{attribute 'linkalways'} 
{attribute 'no_explicit_call' := 'This FB is a CLASS and must be accessed using methods or properties'}
{attribute 'enable_dynamic_creation'}
FUNCTION_BLOCK _TcVnRectangle EXTENDS AliasDatatypeBase
VAR
	localData : TcVnRectangle;
	activeData : REFERENCE TO TcVnRectangle REF= localData;
	aliasBaseDatatype : _TcVnRectangle_DINT;
END_VAR

PROPERTY PUBLIC Address : PVOID
GET
Address := ADR(activeData);
END_GET
END_PROPERTY

METHOD PUBLIC ClearReference
VAR_INPUT
END_VAR
activeData REF= localData;
SetBaseDatatypeReference();
END_METHOD

METHOD PUBLIC Clone : I_Datatype
VAR
    pClone : POINTER TO _TcVnRectangle;
END_VAR
pClone := __NEW(_TcVnRectangle);
Clone := pClone^;
END_METHOD

METHOD FB_init : BOOL
VAR_INPUT
	bInitRetains : BOOL; // if TRUE, the retain variables are initialized (warm start / cold start)
	bInCopyCode : BOOL;  // if TRUE, the instance afterwards gets moved into the copy code (online change)
	//InitialValue : <type>; // if possible, not all values can be initialized
END_VAR
//localData := InitialValue; // if possible, not all values can be initialized
SetBaseDatatypeReference();
AddBaseDatatype(aliasBaseDatatype);
END_METHOD

PROPERTY PUBLIC Identifier : T_MAXSTRING
GET
Identifier := 'TcVnRectangle';
END_GET
END_PROPERTY

METHOD PUBLIC MakeReferenceTo
VAR_INPUT
	ReferenceTarget : REFERENCE TO TcVnRectangle_DINT;
END_VAR
activeData REF= ReferenceTarget;
SetBaseDatatypeReference();
END_METHOD

METHOD PROTECTED SetBaseDatatypeReference
VAR_INPUT
END_VAR
aliasBaseDatatype.MakeReferenceTo(activeData);
END_METHOD

PROPERTY PUBLIC Size : UDINT
GET
Size := SIZEOF(activeData);
END_GET
END_PROPERTY

METHOD TryMakeReferenceTo : BOOL
VAR_INPUT
	Target : I_Datatype;
END_VAR
VAR
	targetAsAlias : I_AliasDatatype;
	pTargetData : POINTER TO TcVnRectangle_DINT;
END_VAR
IF NOT Target.TryResolveAsAliasDatatype(targetAsAlias) THEN
	RETURN;
END_IF

IF targetAsAlias.Identifier <> Identifier THEN
	RETURN;
END_IF

pTargetData := Target.Address;
activeData REF= pTargetData^;
SetBaseDatatypeReference();
TryMakeReferenceTo := TRUE;
END_METHOD

PROPERTY PUBLIC Value : REFERENCE TO TcVnRectangle
GET
Value REF= activeData;
END_GET
END_PROPERTY

END_FUNCTION_BLOCK

(* stored: Version 1.1.0.1, ProductVersion 3.1.4024.13
   POU _TcVnRectangle: Id {66f18127-8e1f-4597-8ea9-6ec469027ad5}, SpecialFunc None
   Folder Core: Id {7ae5aaf7-20cc-0fca-1a98-9f469535e9b6}
   Folder Protected: Id {180266c1-78f1-48ec-9ca5-4c54e7e9deef}
   Folder Customize: Id {68dbbd29-1a5c-04f4-1baa-6b55d9c1ed0c}
   Folder Constructor: Id {d8951580-ae48-4f25-9784-2e9abf3693fc}
   Property Address: Id {a4c6551e-1783-44d5-a59a-fff8e0334b17}
   Get Get: Id {9f714484-433b-4f1b-932e-68d2214c5786}
   Method ClearReference: Id {270244e4-e430-4cdf-9835-ee3b58c92e4d}
   Method Clone: Id {3128c022-9a11-4608-8f9f-2c99a55b4804}
   Method FB_init: Id {0ff46728-fd53-4892-9204-264a3e2557a8}
   Property Identifier: Id {8f895521-f452-4b9d-b139-8ba2ed65a4f6}
   Get Get: Id {6e489654-44c0-4a19-9195-0a16c2cbfb16}
   Method MakeReferenceTo: Id {7449568d-2f56-4bce-b703-855a2e3d7620}
   Method SetBaseDatatypeReference: Id {c449504d-8784-4955-a14a-b966d66ad46f}
   Property Size: Id {038d2981-89c4-4194-a2a6-11bee2b51cf3}
   Get Get: Id {7e13c0aa-87d7-4228-9a3d-83e7f8184a74}
   Method TryMakeReferenceTo: Id {ff161565-760f-49a4-b313-c6389da9febd}
   Property Value: Id {8603c2c7-8a35-449f-a46a-426363d2ac04}
   Get Get: Id {1267fe2b-b097-4424-a8b7-b854de6e686f} *)
